FUNCTION_BLOCK fbIO_AnalogueOutput
VAR_INPUT
END_VAR
VAR_OUTPUT
END_VAR
VAR
END_VAR

END_FUNCTION_BLOCK

(* stored: Version 1.1.0.1, ProductVersion 3.1.4024.11
   POU fbIO_AnalogueOutput: Id {19ccdb33-0c10-46c5-a008-b409d48dd41a}, SpecialFunc None *)
